FUNCTION AddLeadingZeros : STRING
VAR_INPUT
	str : STRING;
	charNumber : USINT;
END_VAR
VAR
END_VAR

AddLeadingZeros := str;
IF charNumber > LEN(str) THEN
	AddLeadingZeros := CONCAT('0', AddLeadingZeros);
	AddLeadingZeros := .AddLeadingZeros(AddLeadingZeros, charNumber);
END_IF

END_FUNCTION

(* stored: Version 1.1.0.1, ProductVersion 3.1.4024.11
   POU AddLeadingZeros: Id {5641fd56-3091-44da-af40-a1a6a765cb15}, SpecialFunc None *)
